{attribute addProperty BoxType "EL5001--0000"}
{attribute addProperty Id "Channel_1AT %I*Channel_7415F5F64050WcStateAT %I*WcState_F855686C1620InfoDataAT %I*InfoData_BC63D37F80100"}
{attribute addProperty CRC "3598405429"}
{attribute addProperty SizeInBites "136"}
{attribute addProperty SizeInBytes "17"}
TYPE EL5001_A4D82738 :
STRUCT
	{attribute addProperty Name "Channel_1"}
	Channel_1 : Channel_7415F5F6;
	{attribute addProperty Name "WcState"}
	WcState : WcState_F855686C;
	{attribute addProperty Name "InfoData"}
	InfoData : InfoData_BC63D37F;
END_STRUCT
END_TYPE

(* stored: Version 1.2.0.0, ProductVersion 3.1.4024.9
   DUT EL5001_A4D82738: Id {22304169-2d13-4a1e-9d1d-a5cf14165219} *)
